// TIA Portal project "CoinChanger" (V16)

(* hardware
DEVICE "S7-1200 station_1"  S7-1200 Station
   slot 0: "Rack_0"  S7-1200 Rack  Rack  V1.0
   slot 1: "PLC_1"  CPU 1214C DC/DC/DC  6ES7 214-1AG31-0XB0  V3.0
   slot 3: "AQ 1x12BIT_1"  AQ1 signal board  6ES7 232-4HA30-0XB0  V1.0
*)

// ===== PLC "PLC_1"  CPU 1214C DC/DC/DC =====

VAR_GLOBAL   // PLC tag table "Default tag table"
   "Qt1" AT %M0.0 : Bool;
   "Dm1" AT %M0.1 : Bool;
   "Qt2" AT %M0.2 : Bool;
   "Req" AT %M0.3 : Bool;
   "Accept" AT %M0.4 : Bool;
   "Dm2" AT %M0.5 : Bool;
   "Change" AT %M0.6 : Bool;
   "Reject" AT %M0.7 : Bool;
END_VAR

ORGANIZATION_BLOCK "Main"   // OB1, LAD, ProgramCycle
TITLE = "Main Program Sweep (Cycle)"
{ S7_Optimized_Access := 'TRUE' }
VERSION : 0.1
BEGIN

REGION Network 1
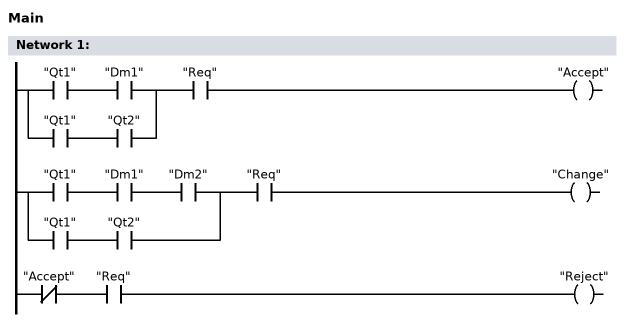
   RUNG wire#powerrail
      Contact( "Qt1" )
      Contact( "Dm1" )
      wire#w1
      Contact( "Req" )
      Coil( "Accept" )
   END_RUNG
   RUNG wire#powerrail
      Contact( "Qt1" )
      Contact( "Qt2" )
   END_RUNG wire#w1
   RUNG wire#powerrail
      Contact( "Qt1" )
      Contact( "Dm1" )
      Contact( "Dm2" )
      wire#w2
      Contact( "Req" )
      Coil( "Change" )
   END_RUNG
   RUNG wire#powerrail
      Contact( "Qt1" )
      Contact( "Qt2" )
   END_RUNG wire#w2
   RUNG wire#powerrail
      I_Contact( "Accept" )
      Contact( "Req" )
      Coil( "Reject" )
   END_RUNG
   // the same network as SCL:
   "Accept" := (("Qt1" AND "Dm1") OR ("Qt1" AND "Qt2")) AND "Req";
   "Change" := (("Qt1" AND "Dm1" AND "Dm2") OR ("Qt1" AND "Qt2")) AND "Req";
   "Reject" := NOT "Accept" AND "Req";
END_REGION
END_ORGANIZATION_BLOCK